// TIA Portal V17 export
// export: Created 2023-04-20T14:56:46.0996566Z, ExportSetting WithDefaults, DisplayName Totally Integrated Automation Portal, DisplayVersion V17, DisplayName TIA Portal Openness, DisplayVersion V17, DisplayName TIA Portal Version Control Interface, DisplayVersion V17, DisplayName STEP 7 Professional, DisplayVersion V17, DisplayName STEP 7 Safety, DisplayVersion V17, DisplayName WinCC Professional, DisplayVersion V17
TYPE "Stack.Interface.UDT"
// stored: Access Published, IsFailsafeCompliant false
   STRUCT
      clear : Bool;
      pop : Bool;
      push : Bool;
      status : String;
      value : Int;
   END_STRUCT;
END_TYPE
